                    11:
                        IF nTestStep = 0 THEN
                            stHMICommand.eCommandType := CMD_MOVE_ABSOLUTE;
                            stHMICommand.nAxisIndex := 1;
                            stHMICommand.fValue1 := 140.0;
                            stHMICommand.fValue2 := 100.0;
                            stHMICommand.bExecute := TRUE;
                            nTestStep := 1;
                        ELSIF (nTestStep = 1) AND (nCyclesInPhase >= 20) THEN
                            GVL_VirtualIO.stVirtualIO.abEncoderHealthy[1] := FALSE;
                            IF (eCurrentMode = MODE_FAULT) AND
                               (NOT astAxisStatus[1].bFeedbackHealthy) THEN
                                bFaultObserved := TRUE;
                                GVL_VirtualIO.stVirtualIO.abEncoderHealthy[1] := TRUE;
                                nTestStep := 2;
                            END_IF
                        ELSIF nTestStep = 2 THEN
                            stHMICommand.eCommandType := CMD_RESET;
                            stHMICommand.bExecute := TRUE;
                            nTestStep := 3;
                        ELSIF nTestStep = 3 THEN
                            nTestStep := 4;
                        ELSIF (nTestStep = 4) AND (nCyclesInPhase >= 100) THEN
                            stHMICommand.eCommandType := CMD_RESET_ALL_ALARMS;
                            stHMICommand.bExecute := TRUE;
                            nTestStep := 5;
                        ELSIF nTestStep = 5 THEN
                            nTestStep := 6;
                        ELSIF (nTestStep = 6) AND (nCyclesInPhase >= 150) THEN
                            stHMICommand.eCommandType := CMD_MODE_REQUEST;
                            stHMICommand.eTargetMode := MODE_MANUAL_JOG;
                            stHMICommand.bExecute := TRUE;
                            nTestStep := 7;
                        ELSIF (nTestStep = 7) AND (eCurrentMode = MODE_MANUAL_JOG) THEN
                            eTestPhase := TEST_VERIFY;
                        END_IF

                    12:
                        IF nTestStep = 0 THEN
                            stHMICommand.eCommandType := CMD_MOVE_ABSOLUTE;
                            stHMICommand.nAxisIndex := 1;
                            stHMICommand.fValue1 := 120.0;
                            stHMICommand.fValue2 := 100.0;
                            stHMICommand.bExecute := TRUE;
                            nTestStep := 1;
                        ELSIF (nTestStep = 1) AND (nCyclesInPhase >= 20) THEN
                            GVL_VirtualIO.stVirtualIO.bEtherCATOK := FALSE;
                            IF (eCurrentMode = MODE_FAULT) AND
                               (NOT stSafetyStatus.bNetworkHealthy) THEN
                                bFaultObserved := TRUE;
                                GVL_VirtualIO.stVirtualIO.bEtherCATOK := TRUE;
                                nTestStep := 2;
                            END_IF
                        ELSIF nTestStep = 2 THEN
                            stHMICommand.eCommandType := CMD_RESET;
                            stHMICommand.bExecute := TRUE;
                            nTestStep := 3;
                        ELSIF nTestStep = 3 THEN
                            nTestStep := 4;
                        ELSIF (nTestStep = 4) AND (nCyclesInPhase >= 90) THEN
                            stHMICommand.eCommandType := CMD_RESET_ALL_ALARMS;
                            stHMICommand.bExecute := TRUE;
                            nTestStep := 5;
                        ELSIF nTestStep = 5 THEN
                            nTestStep := 6;
                        ELSIF (nTestStep = 6) AND (nCyclesInPhase >= 140) THEN
                            stHMICommand.eCommandType := CMD_MODE_REQUEST;
                            stHMICommand.eTargetMode := MODE_MANUAL_JOG;
                            stHMICommand.bExecute := TRUE;
                            nTestStep := 7;
                        ELSIF (nTestStep = 7) AND (eCurrentMode = MODE_MANUAL_JOG) THEN
                            eTestPhase := TEST_VERIFY;
                        END_IF

                    13:
                        IF nTestStep = 0 THEN
                            stHMICommand.eCommandType := CMD_STOP;
                            stHMICommand.nAxisIndex := 1;
                            stHMICommand.bExecute := TRUE;
                            nTestStep := 1;
                        ELSIF nCyclesInPhase >= 30 THEN
                            eTestPhase := TEST_VERIFY;
                        END_IF

                    14:
                        GVL_VirtualIO.stVirtualIO.bEStop := TRUE;
                        GVL_VirtualIO.stVirtualIO.bSafetyRelayFB := TRUE;
                        GVL_VirtualIO.stVirtualIO.bGuardDoorClosed := TRUE;
                        GVL_VirtualIO.stVirtualIO.bSTOHealthy := TRUE;
                        GVL_VirtualIO.stVirtualIO.bEtherCATOK := TRUE;
                        GVL_VirtualIO.stVirtualIO.bWatchdogOK := TRUE;
                        GVL_VirtualIO.stVirtualIO.abDriveReady[1] := TRUE;
                        GVL_VirtualIO.stVirtualIO.abDriveFault[1] := FALSE;
                        GVL_VirtualIO.stVirtualIO.abEncoderHealthy[1] := TRUE;
                        IF nCyclesInPhase >= 30 THEN
                            eTestPhase := TEST_VERIFY;
                        END_IF

                    15:
                        IF nTestStep = 0 THEN
                            GVL_VirtualIO.stVirtualIO.bWatchdogOK := FALSE;
                            IF (eCurrentMode = MODE_FAULT) AND
                               (NOT stSafetyStatus.bWatchdogHealthy) THEN
                                bFaultObserved := TRUE;
                                GVL_VirtualIO.stVirtualIO.bWatchdogOK := TRUE;
                                nTestStep := 1;
                            END_IF
                        ELSIF nTestStep = 1 THEN
                            stHMICommand.eCommandType := CMD_RESET;
                            stHMICommand.bExecute := TRUE;
                            nTestStep := 2;
                        ELSIF nTestStep = 2 THEN
                            nTestStep := 3;
                        ELSIF (nTestStep = 3) AND (nCyclesInPhase >= 80) THEN
                            stHMICommand.eCommandType := CMD_RESET_ALL_ALARMS;
                            stHMICommand.bExecute := TRUE;
                            nTestStep := 4;
                        ELSIF nTestStep = 4 THEN
                            nTestStep := 5;
                        ELSIF (nTestStep = 5) AND (nCyclesInPhase >= 130) THEN
                            stHMICommand.eCommandType := CMD_MODE_REQUEST;
                            stHMICommand.eTargetMode := MODE_MANUAL_JOG;
                            stHMICommand.bExecute := TRUE;
                            nTestStep := 6;
                        ELSIF (nTestStep = 6) AND (eCurrentMode = MODE_MANUAL_JOG) THEN
                            eTestPhase := TEST_VERIFY;
                        END_IF

                    16:
                        IF nTestStep = 0 THEN
                            stHMICommand.eCommandType := CMD_MODE_REQUEST;
                            stHMICommand.eTargetMode := MODE_OFF;
                            stHMICommand.bExecute := TRUE;
                            nTestStep := 1;
                        ELSIF nTestStep = 1 THEN
                            nTestStep := 2;
                        ELSIF (nTestStep = 2) AND (nCyclesInPhase >= 30) THEN
                            stHMICommand.eCommandType := CMD_MOVE_ABSOLUTE;
                            stHMICommand.nAxisIndex := 1;
                            stHMICommand.fValue1 := 50.0;
                            stHMICommand.fValue2 := 100.0;
                            stHMICommand.bExecute := TRUE;
                            nTestStep := 3;
                        ELSIF nCyclesInPhase >= 60 THEN
                            eTestPhase := TEST_VERIFY;
                        END_IF
                END_CASE

                IF nCyclesInPhase > 5000 THEN
                    stTestResult.eResult := TRES_TIMEOUT;
                    sActual := 'Test step exceeded 50 second timeout';
                    eTestPhase := TEST_TEARDOWN;
                END_IF

            TEST_VERIFY:
                IF nVerifyDwellCycles < 5 THEN
                    nVerifyDwellCycles := nVerifyDwellCycles + 1;
                ELSE
                    CASE nCurrentTestID OF
                        1:
                            bVerificationPassed := (eCurrentMode = MODE_MANUAL_JOG) AND
                                astAxisStatus[1].bHomed AND astAxisStatus[2].bHomed;
                            sActual := 'Startup, homing and MANUAL-ready state evaluated';
                        2:
                            bVerificationPassed :=
                                ABS(astAxisStatus[1].fActualPosition - 100.0) <= 0.1;
                            sActual := 'Absolute position tolerance evaluated';
                        3:
                            bVerificationPassed :=
                                ABS(astAxisStatus[1].fActualPosition - fExpectedPosition) <= 0.1;
                            sActual := 'Relative position tolerance evaluated';
                        4:
                            bVerificationPassed := (fPeakPosition > fInitialPosition) AND
                                (fLowPosition < fPeakPosition) AND
                                (NOT astAxisStatus[1].bInMotion);
                            sActual := 'Bidirectional jog displacement and standstill evaluated';
                        5:
                            bVerificationPassed := bFaultObserved AND
                                (eCurrentMode = MODE_MANUAL_JOG) AND stSafetyStatus.bSafeToRun;
                            sActual := 'Positive limit FAULT and recovery evaluated';
                        6:
                            bVerificationPassed := bFaultObserved AND
                                (eCurrentMode = MODE_MANUAL_JOG) AND stSafetyStatus.bSafeToRun;
                            sActual := 'Negative limit FAULT and recovery evaluated';
                        7:
                            bVerificationPassed := bFaultObserved AND
                                (eCurrentMode = MODE_MANUAL_JOG) AND stSafetyStatus.bSafeToRun;
                            sActual := 'E-stop FAULT and recovery evaluated';
                        8:
                            bVerificationPassed := bFaultObserved AND
                                (eCurrentMode = MODE_MANUAL_JOG) AND stSafetyStatus.bSafeToRun;
                            sActual := 'Guard door FAULT and recovery evaluated';
                        9:
                            bVerificationPassed := bFaultObserved AND
                                (eCurrentMode = MODE_MANUAL_JOG) AND
                                (NOT astAxisStatus[1].bError);
                            sActual := 'Drive fault latch and reset evaluated';
                        10:
                            bVerificationPassed := bFaultObserved AND
                                (eCurrentMode = MODE_MANUAL_JOG) AND
                                (NOT astAxisStatus[1].bError);
                            sActual := 'Following error latch and reset evaluated';
                        11:
                            bVerificationPassed := bFaultObserved AND
                                (eCurrentMode = MODE_MANUAL_JOG) AND
                                astAxisStatus[1].bFeedbackHealthy;
                            sActual := 'Encoder feedback loss and reset evaluated';
                        12:
                            bVerificationPassed := bFaultObserved AND
                                (eCurrentMode = MODE_MANUAL_JOG) AND
                                stSafetyStatus.bNetworkHealthy;
                            sActual := 'EtherCAT/network dropout and reset evaluated';
                        13:
                            bVerificationPassed := NOT astAxisStatus[1].bInMotion;
                            sActual := 'Harness established safe standstill for ADS restart';
                        14:
                            bVerificationPassed := GVL_VirtualIO.stVirtualIO.bEStop AND
                                GVL_VirtualIO.stVirtualIO.bSafetyRelayFB AND
                                GVL_VirtualIO.stVirtualIO.bGuardDoorClosed AND
                                GVL_VirtualIO.stVirtualIO.bSTOHealthy AND
                                GVL_VirtualIO.stVirtualIO.bEtherCATOK AND
                                GVL_VirtualIO.stVirtualIO.bWatchdogOK AND
                                GVL_VirtualIO.stVirtualIO.abDriveReady[1] AND
                                (NOT GVL_VirtualIO.stVirtualIO.abDriveFault[1]) AND
                                GVL_VirtualIO.stVirtualIO.abEncoderHealthy[1];
                            sActual := 'Harness established safe defaults for ADS reset';
                        15:
                            bVerificationPassed := bFaultObserved AND
                                (eCurrentMode = MODE_MANUAL_JOG) AND
                                stSafetyStatus.bWatchdogHealthy;
                            sActual := 'Watchdog timeout FAULT and recovery evaluated';
                        16:
                            bVerificationPassed := (NOT astAxisStatus[1].bInMotion) AND
                                (nActiveAlarmCount > 0);
                            sActual := 'Invalid OFF-state move rejection evaluated';
                    END_CASE

                    IF bVerificationPassed THEN
                        stTestResult.eResult := TRES_PASS;
                    ELSE
                        stTestResult.eResult := TRES_FAIL;
                    END_IF
                    eTestPhase := TEST_TEARDOWN;
                END_IF

            TEST_TEARDOWN:
                stTestResult.sActual := sActual;
                stTestResult.tDuration := UDINT_TO_TIME(nCyclesInPhase * 10);
                astTestSummary[nCurrentTestID] := stTestResult;
                nTestsRun := nTestsRun + 1;
                IF stTestResult.eResult = TRES_PASS THEN
                    nTestsPassed := nTestsPassed + 1;
                ELSE
                    nTestsFailed := nTestsFailed + 1;
                END_IF

                GVL_VirtualIO.stVirtualIO.bEStop := TRUE;
                GVL_VirtualIO.stVirtualIO.bSafetyRelayFB := TRUE;
                GVL_VirtualIO.stVirtualIO.bGuardDoorClosed := TRUE;
                GVL_VirtualIO.stVirtualIO.bSTOHealthy := TRUE;
                GVL_VirtualIO.stVirtualIO.bEtherCATOK := TRUE;
                GVL_VirtualIO.stVirtualIO.bWatchdogOK := TRUE;
                GVL_VirtualIO.stVirtualIO.abLimitPos[1] := TRUE;
                GVL_VirtualIO.stVirtualIO.abLimitNeg[1] := TRUE;
                GVL_VirtualIO.stVirtualIO.abDriveReady[1] := TRUE;
                GVL_VirtualIO.stVirtualIO.abDriveFault[1] := FALSE;
                GVL_VirtualIO.stVirtualIO.abEncoderHealthy[1] := TRUE;
                GVL_VirtualIO.stVirtualIO.abFollowingError[1] := FALSE;
                stHMICommand.bExecute := FALSE;

                IF bRunSuite AND (nCurrentTestID < 16) THEN
                    nCurrentTestID := nCurrentTestID + 1;
                    eTestPhase := TEST_SETUP;
                    nTestStep := 0;
                    nCyclesInPhase := 0;
                ELSE
                    eTestPhase := TEST_DONE;
                END_IF

            TEST_DONE:
                bTestSuiteRunning := FALSE;
                bTestSuiteComplete := TRUE;
                bRunSuite := FALSE;
                eTestPhase := TEST_IDLE;
        END_CASE
    END_IF
END_IF

END_FUNCTION_BLOCK
